{attribute 'linkalways'} 
{attribute 'no_explicit_call' := 'This FB is a CLASS and must be accessed using methods or properties'}
{attribute 'enable_dynamic_creation'}
FUNCTION_BLOCK FINAL LE_USINT EXTENDS Node
VAR
	in1 : _USINT(0);
	in2 : _USINT(0);
	out : _BOOL(FALSE);
END_VAR

METHOD PUBLIC Clone : I_Node
VAR
	pNode : POINTER TO LE_USINT;
END_VAR
pNode := __NEW(LE_USINT);
Clone := pNode^;
END_METHOD

METHOD FB_init : BOOL
VAR_INPUT
	bInitRetains : BOOL; // if TRUE, the retain variables are initialized (warm start / cold start)
	bInCopyCode : BOOL;  // if TRUE, the instance afterwards gets moved into the copy code (online change)
END_VAR
AddInput('in1',THIS^.in1);
AddInput('in2',THIS^.in2);
AddOutput('out', THIS^.out);
END_METHOD

METHOD PROTECTED OnExecute
VAR
END_VAR
out.Value := in1.Value <= in2.Value;
END_METHOD

END_FUNCTION_BLOCK

(* stored: Version 1.1.0.1, ProductVersion 3.1.4024.15
   POU LE_USINT: Id {d24d2992-53e7-4a73-844c-d09a517e0c31}, SpecialFunc None
   Folder Constructor: Id {0a12dad8-773d-4c76-a989-c62dc6150f42}
   Method Clone: Id {830e620f-9f25-4872-93f5-65f0f90cd779}
   Method FB_init: Id {e637075c-0058-4b0a-921f-f4688c76fa9e}
   Method OnExecute: Id {f096092c-1050-429c-83bb-38ead3f0e4b5} *)
